FUNCTION_BLOCK PUBLIC FB_TriStableSwitch
VAR_INPUT
	iAnalog		:INT:=0;
END_VAR
VAR_OUTPUT
	bCooling	:BOOL:=FALSE;
	bHeating	:BOOL:=FALSE;
END_VAR
VAR
	iSelector	:INT:=0;
END_VAR

iSelector:=iAnalog/10892;
CASE iSelector OF
	0:
		bCooling:=TRUE;
		bHeating:=FALSE;
	1:
		bCooling:=FALSE;
		bHeating:=FALSE;
	2:
		bCooling:=FALSE;
		bHeating:=TRUE;
END_CASE

END_FUNCTION_BLOCK

(* stored: Version 1.1.0.1, ProductVersion 3.1.4024.4
   POU FB_TriStableSwitch: Id {ae07a299-fc16-477c-8bfa-8572efb31ed1}, SpecialFunc None *)
